FUNCTION_BLOCK Atuador_Coester_CSR6T_HMI (* Service Interface Function Block Type *)
  (* Standard: 61499-2 *)
  (* Version 0.0, 1/26/2026, Schneider Electric, template *)
  PACKAGE Hidryco.HidrycoLib;
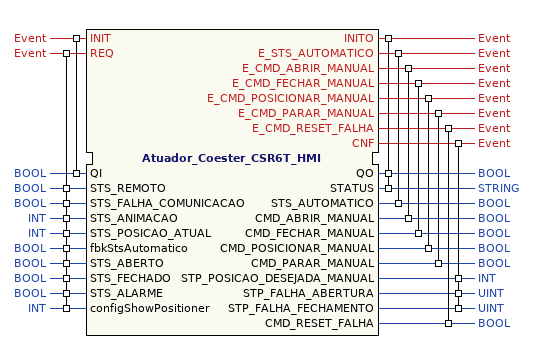
  EVENT_INPUT
    INIT WITH QI;
    REQ WITH STS_REMOTO, STS_ANIMACAO, STS_POSICAO_ATUAL, STS_FALHA_COMUNICACAO, fbkStsAutomatico, STS_ABERTO, STS_FECHADO, STS_ALARME, configShowPositioner;
  END_EVENT
  EVENT_OUTPUT
    INITO WITH QO, STATUS;
    E_STS_AUTOMATICO WITH STS_AUTOMATICO;
    E_CMD_ABRIR_MANUAL WITH CMD_ABRIR_MANUAL;
    E_CMD_FECHAR_MANUAL WITH CMD_FECHAR_MANUAL;
    E_CMD_POSICIONAR_MANUAL WITH CMD_POSICIONAR_MANUAL;
    E_CMD_PARAR_MANUAL WITH CMD_PARAR_MANUAL;
    E_CMD_RESET_FALHA WITH CMD_RESET_FALHA;
    CNF WITH STP_FALHA_ABERTURA, STP_FALHA_FECHAMENTO, STP_POSICAO_DESEJADA_MANUAL;
  END_EVENT
  VAR_INPUT
    QI : BOOL;
    STS_REMOTO : BOOL;
    STS_FALHA_COMUNICACAO : BOOL;
    STS_ANIMACAO : INT;
    STS_POSICAO_ATUAL : INT;
    fbkStsAutomatico : BOOL;
    STS_ABERTO : BOOL; (* Para Nereda *)
    STS_FECHADO : BOOL; (* Para Nereda *)
    STS_ALARME : BOOL; (* Para Nereda *)
    configShowPositioner : INT; (* Alterar a porcentagem de abertura (0 - Only ON OFF, 1 - With Positioner) *)
  END_VAR
  VAR_OUTPUT
    QO : BOOL; (* Event Output Qualifier *)
    STATUS : STRING; (* Service Status *)
    STS_AUTOMATICO : BOOL;
    CMD_ABRIR_MANUAL : BOOL;
    CMD_FECHAR_MANUAL : BOOL;
    CMD_POSICIONAR_MANUAL : BOOL;
    CMD_PARAR_MANUAL : BOOL;
    STP_POSICAO_DESEJADA_MANUAL : INT;
    STP_FALHA_ABERTURA : UINT;
    STP_FALHA_FECHAMENTO : UINT;
    CMD_RESET_FALHA : BOOL;
  END_VAR
  SERVICE /
    SEQUENCE 
    END_SEQUENCE
  END_SERVICE
END_FUNCTION_BLOCK
